TYPE E_LAKESHORE_ERROR :
(
	OK				:= 16#0000,
	NOT_IN_OP_STATE	:= 16#0001,
	NOT_INIT		:= 16#0002,
	TIMEOUT			:= 16#0004,
	COMM			:= 16#0008,
	WRONG_STATE		:= 16#0010,
	NOT_IDLE		:= 16#0020
);
END_TYPE

(* stored: Version 1.1.0.1, ProductVersion 3.1.4022.16
   DUT E_LAKESHORE_ERROR: Id {285603a0-9032-4aa6-9f75-b7e3769b7cd8} *)
